// TIA Portal V20 export
DATA_BLOCK "SyncMotion_Legacy"   // DB448
// stored: Access Published, MemoryReserve 100, Namespace Unit1
   VAR
      General : Struct
         stageWidth : LReal := 244.14;
         stageWidthOffset : LReal := 33.18;
         stageGap : LReal := 1.0;
         stageHeight : LReal := 350.0;
         lineSpeed : LReal;
         startSpeedCpm : LReal := 5.0;
         accTime : LReal := 2.0;
         dccTime : LReal := 2.0;
         countOffset : LReal;
         nowValue : LReal;
         nowCount : DInt;
         stopValue : LReal;
         stopCount : DInt;
         stopTarget : LReal;
         repeatMode : Bool;
         onlyStackMode : Bool;
         anodeToDo : Bool;
         cathodeToDo : Bool;
      END_STRUCT;
      ReelcutInterface : Struct
         anodeReelcutStart : Bool;
         anodeReelcutRunCheck : Bool;
         cathodeReelcutStart : Bool;
         cathodeReelcutRunCheck : Bool;
         stackStop : Bool;
         stackStopCheck : Bool;
         forceStop : Bool;
         forceStopComplete : Bool;
         anodeSize : LReal;
         anodeReelcutPrePosition : LReal;
         anodeReelcutCount : LReal;
         anodeReelcutVelocity : LReal;
         anodeReelcutAcceleration : LReal;
         anodeReelcutDeceleration : LReal;
         anodeStart_anodeRunOffset : LReal;
         anodeStart_cathodeRunOffset : LReal;
         anodeStart_anodeRunTimeOffset : LReal;
         anodeStart_cathodeRunTimeOffset : LReal;
         cathodeSize : LReal;
         cathodeReelcutPrePosition : LReal;
         cathodeReelcutCount : LReal;
         cathodeReelcutVelocity : LReal;
         cathodeReelcutAcceleration : LReal;
         cathodeReelcutDeceleration : LReal;
         cathodeStart_anodeRunOffset : LReal;
         cathodeStart_cathodeRunOffset : LReal;
         cathodeStart_anodeRunTimeOffset : LReal;
         cathodeStart_cathodeRunTimeOffset : LReal;
      END_STRUCT;
      Em0 : Struct
         dancerValueChanged : Bool;
         dancerMode : Int := 2;
         dancerHighKp : LReal := 2.0;
         dancerHighIntegTime : LReal := 0.0;
         dancerHighLimit : LReal := 10.0;
         dancerLowKp : LReal := 0.8;
         dancerLowIntegTime : LReal := 0.0;
         dancerLowLimit : LReal := 5.0;
      END_STRUCT;
      Em1 : Struct
         dancerValueChanged : Bool;
         dancerMode : Int := 1;
         dancerHighKp : LReal := 0.1;
         dancerHighIntegTime : LReal := 0.0;
         dancerHighLimit : LReal := 10.0;
         dancerLowKp : LReal := 0.1;
         dancerLowIntegTime : LReal := 0.0;
         dancerLowLimit : LReal := 5.0;
      END_STRUCT;
      Em2 : Struct
         tmepBit : Bool;
      END_STRUCT;
      Em3 : Struct
         compensatorCamEnabled : Bool;
         unwinderGearEnabled : Bool;
         stackJobCompleteChecked : Bool;
         calculateDiameter : Bool;
         sequenceComplete : Bool;
         stopRequest : Bool;
         stopStart : Bool;
         stopComplete : Bool;
         compensatorOffset : LReal;
         compensatorStart : LReal := 0.0;
         compensatorEnd : LReal := 75.0;
         compensatorStartOffset : LReal;
         preCount : LReal;
         prePosition : LReal;
         targetPosition : LReal;
         PretargetPosition : LReal;
         PreReelCutTargetCount : LReal;
         UnwinderGearRatio : DInt := 10000;
         unwinderDelay : Time;
         CompansatorAutoReadyDis : LReal;
      END_STRUCT;
      Em4 : Struct
         anodePnP1XCamEnabled : Bool;
         anodePnP1ZCamEnabled : Bool;
         anodePnP2XCamEnabled : Bool;
         anodePnP2ZCamEnabled : Bool;
         anodeDownComplete1 : Bool;
         anodeDownComplete2 : Bool;
         anodeSupplyCheck : Bool;
         anodeFinishCheck : Bool;
         anodeSupplyComplete : Bool;
         anodeFinishComplete : Bool;
         anodeReady : Bool;
         anodeRequest : Bool;
         stackJobCompleteChecked : Bool;
         stopRequest : Bool;
         stopComplete : Bool;
         anodePnP1HomePos : Bool;
         anodePnP1WorkPos : Bool;
         anodePnP2HomePos : Bool;
         anodePnP2WorkPos : Bool;
         anodeAvoidPos : Bool;
         anodeReelcutRequest : Bool;
         anodeStartCase : DInt;
         anodePnPXStart : LReal := 0.0;
         anodePnPXEnd : LReal := 75.0;
         anodePnPZDownStart : LReal := 65.0;
         anodePnPZDownEnd : LReal := 75.0;
         anodePnPZUpStart : LReal := 90.0;
         anodePnPZUpEnd : LReal := 100.0;
         anodePnP1ZOnPos : LReal := 5.0;
         anodePnP1ZOffPos : LReal := 5.0;
         anodeReelCutOnPos : LReal := 5.0;
         anodePnP2ZOnPos : LReal := 5.0;
         anodePnP2ZOffPos : LReal := 5.0;
         anodeAlignOnPos : LReal := 5.0;
         anodeAlignOffPos : LReal := 5.0;
         anodeVisionTrigger : LReal := 5.0;
         anodeVisionClean : LReal := 5.0;
      END_STRUCT;
      Em5 : Struct
         cathodePnP1XCamEnabled : Bool;
         cathodePnP1ZCamEnabled : Bool;
         cathodePnP2XCamEnabled : Bool;
         cathodePnP2ZCamEnabled : Bool;
         cathodeDownComplete1 : Bool;
         cathodeDownComplete2 : Bool;
         cathodeSupplyCheck : Bool;
         cathodeFinishCheck : Bool;
         cathodeSupplyComplete : Bool;
         cathodeFinishComplete : Bool;
         cathodeReady : Bool;
         cathodeRequest : Bool;
         stackJobCompleteChecked : Bool;
         stopRequest : Bool;
         stopComplete : Bool;
         cathodePnP1HomePos : Bool;
         cathodePnP1WorkPos : Bool;
         cathodePnP2HomePos : Bool;
         cathodePnP2WorkPos : Bool;
         cathodeAvoidPos : Bool;
         cathodeReelcutRequest : Bool;
         cathodeStartCase : DInt;
         cathodePnPXStart : LReal := 0.0;
         cathodePnPXEnd : LReal := 75.0;
         cathodePnPZDownStart : LReal := 65.0;
         cathodePnPZDownEnd : LReal := 75.0;
         cathodePnPZUpStart : LReal := 90.0;
         cathodePnPZUpEnd : LReal := 100.0;
         cathodePnP1ZOnPos : LReal := 5.0;
         cathodePnP1ZOffPos : LReal := 5.0;
         cathodeReelCutOnPos : LReal := 5.0;
         cathodePnP2ZOnPos : LReal := 5.0;
         cathodePnP2ZOffPos : LReal := 5.0;
         cathodeAlignOnPos : LReal := 5.0;
         cathodeAlignOffPos : LReal := 5.0;
         cathodeVisionTrigger : LReal := 5.0;
         cathodeVisionClean : LReal := 5.0;
      END_STRUCT;
      Em6 : Struct
         finalRollerCamEnabled : Bool;
         mandrelAnodeFrontYCamEnabled : Bool;
         mandrelAnodeFrontZCamEnabled : Bool;
         mandrelAnodeRearYCamEnabled : Bool;
         mandrelAnodeRearZCamEnabled : Bool;
         mandrelCathodeFrontYCamEnabled { ExternalVisible := 'False'} : Bool;
         mandrelCathodeFrontZCamEnabled : Bool;
         mandrelCathodeRearYCamEnabled : Bool;
         mandrelCathodeRearZCamEnabled : Bool;
         finalRollerMove : Bool;
         finalRollerMoveComplete : Bool;
         anodeGripComplete1 : Bool;
         anodeGripComplete2 : Bool;
         anodeGripComplete3 : Bool;
         cathodeGripComplete1 : Bool;
         cathodeGripComplete2 : Bool;
         cathodeGripComplete3 : Bool;
         finalRollerAnodePos : Bool;
         finalRollerCathodePos : Bool;
         stackStart : Bool;
         stackComplete : Bool;
         stackUpComplete : Bool;
         stackUngripComplete : Bool;
         stackGripComplete : Bool;
         onlyStackComplete : Bool;
         dancerHigh1 : Bool;
         dancerHigh2 : Bool;
         dancerHigh3 : Bool;
         dancerHigh4 : Bool;
         dancerLow1 : Bool;
         dancerLow2 : Bool;
         dancerLow3 : Bool;
         dancerLow4 : Bool;
         stopRequest : Bool;
         stopComplete : Bool;
         anodeSupplyRequest1 : Bool;
         anodeSupplyRequest2 : Bool;
         anodeFinishRequest : Bool;
         anodeSupplyCompleteCheck1 : Bool;
         anodeSupplyCompleteCheck2 : Bool;
         anodeFinishCompleteCheck : Bool;
         cathodeSupplyRequest1 : Bool;
         cathodeSupplyRequest2 : Bool;
         cathodeFinishRequest : Bool;
         cathodeSupplyCompleteCheck1 : Bool;
         cathodeSupplyCompleteCheck2 : Bool;
         cathodeFinishCompleteCheck : Bool;
         startCountCheck : DInt;
         finalRollerStart : LReal := 0.0;
         finalRollerEnd : LReal := 75.0;
         finalRollerDistance : LReal;
         mandrelBwdStartPos : LReal := 75.0;
         mandrelBwdEndPos : LReal := 82.5;
         mandrelFwdStartPos : LReal := 82.5;
         mandrelFwdEndPos : LReal := 90.0;
         mandrelUpStartPos : LReal := 75.0;
         mandrelUpEndPos : LReal := 82.5;
         mandrelDownStartPos : LReal := 87.0;
         mandrelDownEndPos : LReal := 90.0;
         outputCamOffset : LReal := 10.0;
         visionPosOffset : LReal := 0.0;
         visionTime : LReal := 50.0;
      END_STRUCT;
      Em7 : Struct
         unloadGripComplete : Bool;
         unloadClampLockComplete : Bool;
         unloadClampCuttingComplete : Bool;
         unloadJobComplete : Bool;
         radius : LReal := 122.07;
         sepaDistances : LReal := 976.56;
      END_STRUCT;
   END_VAR
BEGIN
END_DATA_BLOCK
